FUNCTION F_ITC_SendERR : BOOL
(**************************************************************************************
 * 	Application		:	BoxControl Framework
 *	Revision		:	$Revision: 404529 $
 *	Revision date	:	$Date: 2018-04-23 08:21:38 +0200 (Mo., 23 Apr 2018) $
 *	Last changed by	:	$Author: b7bolm $
 *	URL				:	$URL: http://almscdc.swisslog.com/repo/SWPD/Development/BoxControlFramework/20_Release/trunk/01_Software/BCF/BCF/JumpStart/20_Product/10_App/11_Com/10_Lib/10_Conv/11_ITC/F_ITC_SendERR.TcPOU $
 *
 *	Purpose			:	Wrap message - ERR
 *
 * ------------------------------------------------------------------------------------
 *	Copyright Swisslog [IP AG], Switzerland. All rights reserved.
 * 
 * ------------------------------------------------------------------------------------
 *	
 * 	Revision History: 
 *
 * 	VERSION			DATE			INITIALS			DESCRIPTION
 *	0.1				01.01.2001		swl					Example
 *
 **************************************************************************************)
VAR_INPUT
	eChannelSrc		: E_MFCS_Channel; // Source communicaton channel
	PositionName	: STRING(Conveyor.POSITION_STRINGLENGTH); // SIS MM-GGG-EEEE-FF-Z
	Code			: INT; // Error type code
	eReturnCode		: E_ErrorConv; // Return code
END_VAR
VAR
	ERR				: ST_ITC_ERR; 
END_VAR

// Map values
ERR.Position := PositionName;
ERR.Code := Code;
ERR.ReturnCode := eReturnCode;

// Forward to ITC
F_ITC_SendERR := fbITC_Manager.M_SendData(
					meChannel	:= eChannelSrc,
					mMsgType	:= E_ITC_MsgTypeConv.E_ERROR_REPORT,
					mpData		:= ADR(ERR),
					mLen		:= SIZEOF(ERR));

END_FUNCTION

(* stored: Version 1.1.0.1, ProductVersion 3.1.4022.12
   POU F_ITC_SendERR: Id {7194bfca-732d-44e1-a508-740602a885d5}, SpecialFunc None *)
